SUBAPPLICATION Uebung_035a3_AX (* Ampelschaltung Österreich (AX) mit Blinker *)
  (* Standard: 61499-2; Description: Copyright (c) 2023 Meisterschulen am Ostbahnhof This program and the accompanying materials are made available under the terms of the Eclipse Public License 2.0 which is available at https://www.eclipse.org/legal/epl-2.0/ SPDX-License-Identifier: EPL-2.0 *)
  (* Version 1.0, 2026-02-01, Franz Höpfinger, Meisterschulen am Ostbahnhof, initial API and implementation and/or initial documentation *)
  PACKAGE Uebungen;
  IMPORT logiBUS::io::DI::logiBUS_DI::Input_I1;
  IMPORT logiBUS::io::DQ::logiBUS_DO::Output_Q1;
  IMPORT logiBUS::io::DQ::logiBUS_DO::Output_Q2;
  IMPORT logiBUS::io::DQ::logiBUS_DO::Output_Q3;
  IMPORT logiBUS::io::DI::logiBUS_DI_Events::BUTTON_SINGLE_CLICK;
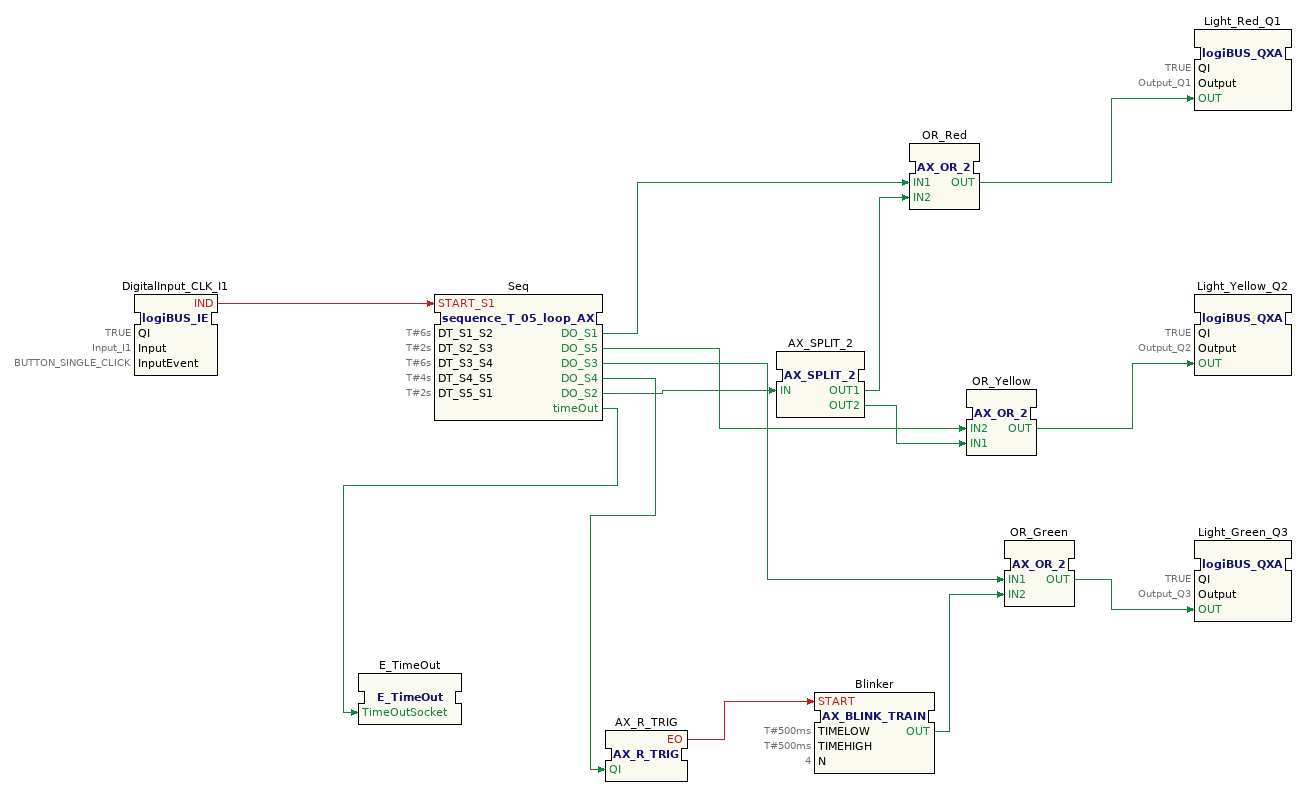
  FBS
    Seq : logiBUS::utils::sequence::timed::sequence_T_05_loop_AX(DT_S1_S2 := T#6s, DT_S2_S3 := T#2s, DT_S3_S4 := T#6s, DT_S4_S5 := T#4s, DT_S5_S1 := T#2s);
    Light_Red_Q1 : logiBUS::io::DQ::logiBUS_QXA(QI := TRUE, Output := Output_Q1);
    Light_Yellow_Q2 : logiBUS::io::DQ::logiBUS_QXA(QI := TRUE, Output := Output_Q2);
    Light_Green_Q3 : logiBUS::io::DQ::logiBUS_QXA(QI := TRUE, Output := Output_Q3);
    Blinker : adapter::events::unidirectional::signals::AX_BLINK_TRAIN(TIMELOW := T#500ms, TIMEHIGH := T#500ms, N := 4);
    OR_Red : adapter::booleanOperators::AX_OR_2;
    OR_Yellow : adapter::booleanOperators::AX_OR_2;
    OR_Green : adapter::booleanOperators::AX_OR_2;
    DigitalInput_CLK_I1 : logiBUS::io::DI::logiBUS_IE(QI := TRUE, Input := Input_I1, InputEvent := BUTTON_SINGLE_CLICK);
    AX_R_TRIG : adapter::events::unidirectional::AX_R_TRIG;
    AX_SPLIT_2 : adapter::events::unidirectional::AX_SPLIT_2;
    E_TimeOut : iec61499::events::E_TimeOut;
  END_FBS
  EVENT_CONNECTIONS
    DigitalInput_CLK_I1.IND TO Seq.START_S1;
    AX_R_TRIG.EO TO Blinker.START;
  END_CONNECTIONS
  ADAPTER_CONNECTIONS
    Seq.DO_S1 TO OR_Red.IN1;
    AX_SPLIT_2.OUT1 TO OR_Red.IN2;
    Seq.DO_S5 TO OR_Yellow.IN2;
    Seq.DO_S3 TO OR_Green.IN1;
    Blinker.OUT TO OR_Green.IN2;
    OR_Red.OUT TO Light_Red_Q1.OUT;
    OR_Yellow.OUT TO Light_Yellow_Q2.OUT;
    OR_Green.OUT TO Light_Green_Q3.OUT;
    Seq.DO_S4 TO AX_R_TRIG.QI;
    Seq.DO_S2 TO AX_SPLIT_2.IN;
    AX_SPLIT_2.OUT2 TO OR_Yellow.IN1;
    Seq.timeOut TO E_TimeOut.TimeOutSocket;
  END_CONNECTIONS
END_SUBAPPLICATION
